Staubli VAL3: check_cube.pgx

public program check_cube(tool x_tTool, bool& x_bCheck[])
  local point l_pPoint
  local bool l_bPositive
  local bool l_bNegative
begin
  //
  // CHECK IF THE TOOL IS INSIDE
  //
  x_bCheck=false
  //
  if bCreate_cube
    l_pPoint=here(x_tTool,fCube)
    // check if inside
    // x y z
    if l_pPoint.trsf.z>=-0.1 and l_pPoint.trsf.z<=nDistanceZ_cube
      // check if positive or negative of Y
      l_bPositive=l_pPoint.trsf.y>=-0.1 and l_pPoint.trsf.y<=nDistanceY_cube+0.1 and nDistanceY_cube>=-0.1
      l_bNegative=l_pPoint.trsf.y<=0.1 and l_pPoint.trsf.y>=nDistanceY_cube-0.1 and nDistanceY_cube<=0.1
      if l_bPositive or l_bNegative
        // check if positive or negative of X
        l_bPositive=l_pPoint.trsf.x>=-0.1 and l_pPoint.trsf.x<=nDistanceX_cube+0.1 and nDistanceX_cube>=-0.1
        l_bNegative=l_pPoint.trsf.x<=0.1 and l_pPoint.trsf.x>=nDistanceX_cube-0.1 and nDistanceX_cube<=0.1
        if l_bPositive or l_bNegative
          // is inside
          x_bCheck=true
        endIf
      endIf
    endIf
  endIf
end
